# B&R Automation Studio project CombinedLinenSoiledA9KAN (part 4)

#### zzuld_3Cyclic.ab
```automation-basic
PROGRAM _CYCLIC
   	(* cyclic program *)

	;Unloading Programs 3 - Search and give Destination (Using Bag)

	;----------------------------------------
	;Version 1.00 03/12/2005 D.J. First Issue
	;----------------------------------------
	;Init Sequence
	;-------------

	;Spare Step
	IF (UldStep = 0) THEN
		UldStep = 1
	ENDIF

	;UldStep 1	- Check no bags in Storage are allocated with a destination
	IF (UldStep = 1) THEN

		;Allow next Discharger to search
		R_TRIG(NOT Std.BagsWithDestinations,PLS)
		IF PLS THEN
			Discharger 	= (LastDischarger + 1)
			ScanCount 	= 0
		ENDIF

		;Set ScanCount as alternating Value 25 is about 5 seconds
		IF Std.BagsWithDestinations  OR (ScanCount = 1) THEN
			Discharger 	= (Discharger + 1)
			ScanCount 	= 0
		ENDIF

		ScanCount = (ScanCount + 1)

		IF ((Discharger > EndDischarger) OR (Discharger < StartDischarger))  THEN
			Discharger 	= StartDischarger
		ENDIF

		;Set discharger number in TestDischarger if required
		IF (TestDischarger > 0) THEN
			Discharger = TestDischarger
		ENDIF

		;Read Program Variables
		n = RegOffset[Discharger]

		ProgramStep 			= D[1 + n]
		ProgQtyComplete			= D[2 + n]
		AutoRecirculation 		= (D[1003] = 1)		;Use if Re-cirulation or Offgoing Batching Loop
		RecirculationMaxDepth 	= D[1004]

		ManualLine       		= D[7 + n]
		ManualBags       		= D[8 + n]
		StepsSearched			= D[9 + n]
		SkipIncompleteStep 		= (D[10 + n] = 1)
		AutoRepeat				= (D[11 + n] = 1)
		MixCategories 			= (D[12 + n] = 1)	;Batch must be same category?
		MixCustomers 			= (D[13 + n] = 1) 	;Batch must be same customer?
		NoBagAvailable			= (D[14 + n] = 1)	;Alarm 'No Bag Available'
		ProgramFinished			= (D[15 + n] = 1)	;Alarm 'Finished Program'
		ManualLineRecirc 		= D[1016]
		ManualBagsRecirc 		= D[1017]
		ProgramRunning			= (D[19 + n] = 1)	;Run from TrackView
		ExpressLine 			= D[20 + n]
		CustomerMode			= D[21 + n]			;Customer Mode 0 = Normal Manual, 1 = Reset Pointer on every step, 2 = Check all steps before changing
		ProgramReset			= (D[22 + n] = 1)	;Customer FIFO Reset

		DischargerReady			= Uld[Discharger].SDCReady
		DischargerSpaces		= Line[BufferLineNum[Discharger]].SpaceBIT
		RecircSpaces			= Line[BufferLineNum[EndDischarger + 1]].SpaceBIT

		IF (NOT Std.BagsWithDestinations AND (Discharger > 0)) THEN
			UldStep = 2
		ELSE
			;Allow program to skip blank steps when Bags Have Destinations
			UnusedStep		= (D[40 + n + ProgramStep] = 0) ;Bags = 0
			IF UnusedStep THEN
				UldStep = 15
			ENDIF
		ENDIF

		;If program is new then Clear Search Values
		IF ProgramReset THEN
			Uld[Discharger].FIFOCustomer 		= 0	;Clear Current Customer - FIFO Will allocate next
			Uld[Discharger].LastCustQtyComplete = 0	;Clear Last Quantity
			StepsSearched 						= 0	;Clear Steps Searched / Failed
			D[22 + n]	 						= 0 ;Clear Program Reset
			UldStep 							= 0	;Keep Unloading Step at 0 to allow Customer FIFO to allocate next Customer
		ENDIF

	ENDIF

	;UldStep 2	- Check for a Manual Re-circulation regardless of Discharger
	;			- Note will stop all unloading progrms if not ready
	IF (UldStep = 2) THEN
		IF ((ManualLineRecirc >= StartLineSearch) AND (ManualLineRecirc <= EndLineSearch) AND (ManualBagsRecirc > 0)) THEN
			IF Uld[EndDischarger + 1].SDCReady THEN
				UldStep = 21
			ELSE
				UldStep = 0
			ENDIF
		ELSE
			UldStep = 3
		ENDIF
	ENDIF

	;UldStep 3	- Check Discharger is Ready
	IF (UldStep = 3) THEN
		IF (DischargerReady AND ProgramRunning AND (DischargerSpaces > 0)) THEN
			UldStep = 4
		ELSE
			;If not ready then clear steps searched
			UldStep = 0
		ENDIF
	ENDIF

	;UldStep 4	- Check for a Manual Bags
	IF (UldStep = 4) THEN
		IF ((ManualLine >= StartLineSearch) AND (ManualLine <= EndLineSearch) AND (ManualBags > 0)) THEN
			UldStep = 22
		ELSE
			UldStep = 5
		ENDIF
	ENDIF

	;STEP 5	- Check Express Line
	IF (UldStep = 5) THEN
		IF (ExpressLine > 0) THEN
			ExpressBag  = Line[ExpressLine].FirstBag
		ENDIF
		IF ((Bag[ExpressBag].Cat > 0) AND (ExpressLine > 0) AND (Line[BufferLineNum[Discharger]].SpaceBIT > 0)) THEN
			UldStep = 23
		ELSE
			UldStep = 6
		ENDIF
	ENDIF

	;UldStep 6	- Check Program step
	IF (UldStep = 6) THEN

		;Check if UldStep Valid
		IF (ProgramStep < 1) OR (ProgramStep > 20) THEN
			ProgramStep = 1 					;Set to UldStep 1
			ProgQtyComplete = 0 				;Clear Qty Completed
			IF (CustomerMode = 1) THEN
				Uld[Discharger].FIFOCustomer = 0
			ENDIF
		ENDIF

		UldStep = 7

	ENDIF

	;UldStep 7 - Check for remaining bags on the current Step
	IF (UldStep = 7) THEN

		BatchSize 		= D[80 + n + ProgramStep]
		Quantity 		= D[40 + n + ProgramStep] ;* BatchSize ;Take bags * BatchSize
		BagsRemaining 	= (Quantity - ProgQtyComplete)

		IF ((BagsRemaining > 0) AND (BagsRemaining >= BatchSize)) THEN
			UldStep = 8
		ELSE
			UldStep = 15 ;Step Not Complete Or No Qty
		ENDIF

	ENDIF

	;UldStep 8 - Check the 'Batch' Will fit onto the Buffer
	IF (UldStep = 8) THEN

		BatchSize 		= D[80 + n + ProgramStep]

		IF (DischargerSpaces >= BatchSize) THEN
			UldStep = 9
		ELSE
			UldStep = 0
		ENDIF

	ENDIF

	;UldStep 9 - Set Search Values
	IF (UldStep = 9) THEN

		IF (PriorityLine = 0) THEN
			StartLine = (Uld[Discharger].DischargerStartLine + 1)
			IF ((StartLine < StartLineSearch) OR (StartLine > EndLineSearch)) THEN
				StartLine = StartLineSearch
			ENDIF
		ELSE
			StartLine = PriorityLine
		ENDIF

		SearchLine   = D[60 + n + ProgramStep]
		BatchSize    = D[80 + n + ProgramStep]

		SearchCat[1] = D[100 + n + ProgramStep]
		SearchCat[2] = D[120 + n + ProgramStep]
		SearchCat[3] = D[140 + n + ProgramStep]

		IF (CustomerMode = 0) THEN
			SearchCus[1] = D[181 + n]					;Manually Selected Customer
		ELSE
			SearchCus[1] = Uld[Discharger].FIFOCustomer ;Automatic FIFO Customer Selection
		ENDIF

		SearchSpaces = 0 ;Search Always starts with no spaces on the recirc

		UldStep = 10

	ENDIF

	;UldStep 10 - Search for Bag(s) could be modified to run over several scans to reduce its load on the PLC
	;			  To find the best pos using set RecircSpaces low increasing to max.
	IF (UldStep = 10) THEN

		LOOP FindBest = 1 TO 3 DO

			;Clear the Search Array and Set Depth Allowed 1 for upto 49 storage lines
			FoundLine = 0
			memset(ADR(FoundBag[0]),0,10)
			memset(ADR(LineDepthAllowed[0]),1,50)

			RecircSpacesRemain = SearchSpaces

			IF (FindBest = 1) THEN
				MatchCat1Cus1 = TRUE
				MatchCat2Cus1 = FALSE
				MatchCat3Cus1 = FALSE
			ELSE IF (FindBest = 2) THEN
				MatchCat1Cus1 = MixCategories
				MatchCat2Cus1 = TRUE
				MatchCat3Cus1 = FALSE
			ELSE
				MatchCat1Cus1 = MixCategories
				MatchCat2Cus1 = MixCategories
				MatchCat3Cus1 = TRUE
			ENDIF

			;Loop around all the storage lins row by row.
			LOOP CurrentDepth = 1 TO UnloadingMaxDepth DO ;Always search to max depth to check scan time

				CurrentLine = StartLine

				LOOP LinesSearched = StartLineSearch TO EndLineSearch DO ;Loop around each line

					CurrentBag = (Line[CurrentLine].FirstBag + (CurrentDepth - 1))

					;Search / Add
					;------------
					;For Unloading by line - If there is a bag on the line and the 1st Category = 0 then check Customer valid
					;eg if the 1st Cat and 1st Cus are set to 0 then this would set "CatCusValid" to TRUE but the line must also match
					;Unloading by Customer only cannot be done.

					CusValid = FALSE
					CatValid = FALSE

					;Check the Customer is valid
					IF (Bag[CurrentBag].Cus = SearchCus[1]) THEN
						CusValid = TRUE
					ELSE IF ((SearchCus[1] = 0) AND (CustomerMode = 0)) THEN ;Only Valid If Manual Customer Selection
						CusValid = TRUE
					ENDIF

					;Check the Category is valid
					IF (MatchCat1Cus1 AND (Bag[CurrentBag].Cat = SearchCat[1]) AND (SearchCat[1] > 0)) THEN
						CatValid = TRUE
					ENDIF
					IF (MatchCat2Cus1 AND (Bag[CurrentBag].Cat = SearchCat[2]) AND (SearchCat[2] > 0)) THEN
						CatValid = TRUE
					ENDIF
					IF (MatchCat3Cus1 AND (Bag[CurrentBag].Cat = SearchCat[3]) AND (SearchCat[3] > 0)) THEN
						CatValid = TRUE
					ENDIF
					;If Unloading by line and no Category is set then Set Valid
					IF ((Bag[CurrentBag].Cat > 0) AND (SearchCat[1] = 0) AND (SearchLine > 0)) THEN
						CatValid = TRUE
					ENDIF

					LineValid = ((SearchLine = CurrentLine) OR (SearchLine = 0))

					DepthValid	= ((LineDepthAllowed[CurrentLine] + RecircSpacesRemain) >= CurrentDepth)
					DepthValid2	= ((CurrentDepth <= RecirculationMaxDepth) OR NOT AutoRecirculation)

					IF (CatValid AND CusValid AND LineValid AND DepthValid AND DepthValid2) THEN

						IF (FoundBag[0] < BatchSize)  THEN
							FoundBag[0] = FoundBag[0] + 1
							x 			= FoundBag[0]
							FoundBag[x] = CurrentBag
							FoundLine	= CurrentLine

							;If bags need to go to recirc then dec
							IF (LineDepthAllowed[CurrentLine] < USINT(CurrentDepth)) THEN
								SpacesUsed 			= USINT(CurrentDepth) - LineDepthAllowed[CurrentLine]
								RecircSpacesRemain 	= (RecircSpacesRemain - SpacesUsed)
							ENDIF

							LineDepthAllowed[CurrentLine] = USINT(CurrentDepth + 1)

						ENDIF

					ENDIF

					;-------------
					;End of Search
					;-------------

					;If searching using priority line then start from the Discharger Start Line
					IF CurrentLine = PriorityLine THEN
						CurrentLine = (Uld[Discharger].DischargerStartLine)
					ENDIF

					;Set Next Line
					CurrentLine = (CurrentLine + 1)
					IF CurrentLine > EndLineSearch THEN
						CurrentLine = StartLineSearch
					ENDIF

					;If the new line = priority line then skip as its already been searched
					IF CurrentLine = PriorityLine THEN
						CurrentLine = (CurrentLine + 1)
						IF CurrentLine > EndLineSearch THEN
							CurrentLine = StartLineSearch
						ENDIF
					ENDIF

				ENDLOOP

			ENDLOOP

			EXITIF FoundBag[0] = BatchSize

		ENDLOOP				;Find Best

		;Check if the bags were found
		IF FoundBag[0] = BatchSize THEN
			UldStep = 14 	;Action Results
		ELSE IF (AutoRecirculation AND (SearchSpaces < RecircSpaces)) THEN
			;If recirculation - to find the best possible result inc the search spaces each scan
			;until total spaces searched
			SearchSpaces = (SearchSpaces + 1)
			UldStep = 10	;Try with more recirculation space
		ELSE
			UldStep = 15	;Search Failed
		ENDIF

	ENDIF

	;UldStep 14 - Search Valid give bags destinations, inc qty taken by batchsize
	IF (UldStep = 14) THEN

		LOOP Dest = 1 TO BatchSize DO
			Bag[FoundBag[Dest]].Dst = USINT(BufferLineNum[Discharger])
		ENDLOOP
		ProgQtyComplete = ProgQtyComplete + BatchSize	;Inc Qty Completed
		StepsSearched = 0 								;Clear the search failed UldStep counter
		NoBagAvailable = FALSE 							;No Bags Alarm (OFF)
		LastDischarger = Discharger

		IF AutoRecirculation THEN
			UldStep = 24		;Set Any Bags for Auto-Reirculation
		ELSE
			UldStep = 0
		ENDIF

		;Mode 2 Needs to keep the Qty completed for the next customer
		Uld[Discharger].LastCustQtyComplete = ProgQtyComplete

	ENDIF

	;UldStep 15 - Search Failed
	IF (UldStep = 15) THEN

		BatchSize 		= D[80 + n + ProgramStep]
		;Quantity 		= D[40 + n + ProgramStep] * BatchSize ;Take bags * BatchSize
		Quantity		= (D[40 + n + ProgramStep])
		BagsRemaining 	= (Quantity - ProgQtyComplete)
		UnusedStep		= (D[40 + n + ProgramStep] = 0) ;Bags = 0

		;Inc Steps searched counter
		IF (StepsSearched < 21) THEN
			StepsSearched = (StepsSearched + 1)
		ENDIF

		IF (CustomerMode = 0) THEN
			IF (BagsRemaining = 0) THEN
				UldStep = 16			;Try Next Step
			ELSE IF (SkipIncompleteStep OR UnusedStep) THEN
				UldStep = 16			;Try Next Step
			ELSE
				NoBagAvailable = TRUE 	;Set Alarm and Wait for Operator to change Program or More Bags
				UldStep = 0
			ENDIF
		ENDIF

		IF (CustomerMode = 1) THEN
			IF (BagsRemaining = 0) THEN
				UldStep = 16			;Try Next Step
			ELSE IF (NOT UnusedStep) THEN
				IF (Uld[Discharger].FIFONextCustomer > 0) THEN
					;Mode 1 Search again with the Next Customer Without Changing Step
					Uld[Discharger].FIFOCustomer = Uld[Discharger].FIFONextCustomer
					UldStep = 0
				ELSE
					;Last customer was not found reset FIFO position to 1 and keep searching
					Uld[Discharger].FIFOCustomer = 0 ;Reset the First Customer
					NoBagAvailable = TRUE
					UldStep = 0
				ENDIF
			ELSE IF (SkipIncompleteStep OR UnusedStep) THEN
				UldStep = 16			;Try Next Step
			ELSE
				NoBagAvailable = TRUE	;Set Alarm and Wait for Operator to change Program or More Bags
				UldStep = 0
			ENDIf
		ENDIF

		IF (CustomerMode = 2) THEN
			IF (BagsRemaining = 0) THEN
				UldStep = 16			;Try Next Step
			ELSE IF (StepsSearched = 21) THEN
				IF (Uld[Discharger].FIFONextCustomer > 0) THEN
					;Mode 2 Customer Change Only After 21 Steps Searched
					Uld[Discharger].FIFOCustomer = Uld[Discharger].FIFONextCustomer
					ProgQtyComplete = Uld[Discharger].LastCustQtyComplete
					StepsSearched = 0 ;FREI Use -1 to go to next step
					UldStep = 0
				ELSE
					;Last customer was not found reset FIFO position to 1 and keep searching
					Uld[Discharger].FIFOCustomer = 0 ;Reset the First Customer
					NoBagAvailable = TRUE
					StepsSearched = 0
					UldStep = 0
				ENDIF
			ELSE IF (SkipIncompleteStep OR UnusedStep) THEN
				UldStep = 16			;Try Next Step
			ELSE
				NoBagAvailable = TRUE	;Set Alarm and Wait for Operator to change Program or More Bags
				UldStep = 0
			ENDIF
		ENDIF

	ENDIF

	;Skip Program Step or Set to 1
	IF (UldStep = 16) THEN
		IF (ProgramStep = 20) THEN
			IF AutoRepeat THEN
				ProgramStep = 1
				IF (CustomerMode = 1) THEN
					Uld[Discharger].FIFOCustomer = 0 ;Start Search With First Customer
				ENDIF
			ELSE
				ProgramFinished = TRUE
			ENDIF
		ELSE
			ProgramStep = ProgramStep + 1
			IF (CustomerMode = 1) THEN
				Uld[Discharger].FIFOCustomer = 0 ;Start Search With First Customer
			ENDIF
		ENDIF
		ProgQtyComplete = 0
		UldStep = 0
	ENDIF

	;UldStep 21 -	Manual Bags Recirc
	IF (UldStep = 21) THEN

		CurrentBag = Line[ManualLineRecirc].FirstBag

		IF Bag[CurrentBag].Cat > 0 THEN
			Bag[CurrentBag].Dst = USINT(BufferLineNum[EndDischarger + 1])	;Set Destination
			ManualBagsRecirc    = (ManualBagsRecirc - 1)					;Dec manual bags by 1
		ENDIF

		UldStep = 0

	ENDIF

	;UldStep 21 - Manual Bags to Discharger
	IF (UldStep = 22) THEN

		CurrentBag = Line[ManualLine].FirstBag

		IF Bag[CurrentBag].Cat > 0 THEN
			Bag[CurrentBag].Dst = USINT(BufferLineNum[Discharger])
			ManualBags 			= (ManualBags - 1)				;Dec manual bags by 1
		ENDIF

		UldStep = 0

	ENDIF

	;UldStep 23 - Express Line
	IF (UldStep = 23) THEN

		Bag[ExpressBag].Dst = USINT(BufferLineNum[Discharger])

		UldStep = 0

	ENDIF

	;UldStep 24 - Set Bags to re-circulation line if they need to move out of the way of bags with destinations
	IF (UldStep = 24) THEN

		LOOP CurrentLine = StartLineSearch to EndLineSearch DO
			LOOP CurrentBag = Line[CurrentLine].LastBag DOWNTO Line[CurrentLine].FirstBag DO

				IF (Bag[CurrentBag].Dst > 0) AND (Bag[CurrentBag - 1].Dst = 0) AND (CurrentBag > Line[CurrentLine].FirstBag) THEN
					Bag[CurrentBag - 1].Dst = USINT(BufferLineNum[EndDischarger + 1])
				ENDIF

			ENDLOOP
		ENDLOOP

		UldStep = 0

	ENDIF

	;Outputs
	;-------

	D[1 + n] 		= ProgramStep
	D[2 + n]		= ProgQtyComplete
	D[8 + n] 		= ManualBags
	D[9 + n]		= StepsSearched

	;No bag available is displayed if 20 steps have been searched and program is running
	IF (NoBagAvailable AND ProgramRunning) THEN
		D[14 + n] = 1
		Alarm[Discharger + 100].On		= TRUE
		Alarm[Discharger + 100].Bag 	= 0
		Alarm[Discharger + 100].Name 	= almUldNoBag
		Alarm[Discharger + 100].Beacon	= FALSE
	ELSE
		D[14 + n]	= 0
	ENDIF

	;Program is only finished if on step 20 and Program Running
	IF (ProgramFinished AND ProgramRunning AND (ProgramStep = 20)) THEN
		D[15 + n]	= 1
		Alarm[Discharger + 100].On		= TRUE
		Alarm[Discharger + 100].Bag 	= 0
		Alarm[Discharger + 100].Name 	= almUldProgFinished
		Alarm[Discharger + 100].Beacon	= FALSE
	ELSE
		D[15 + n]	= 0
	ENDIF

	;If no unloading alarms then clear unloading alarm
	IF (D[14 + n] = 0) AND (D[15 + n] = 0) THEN
		Alarm[Discharger + 100].On		= FALSE
		Alarm[Discharger + 100].Bag 	= 0
		Alarm[Discharger + 100].Name 	= almNoAlarm
		Alarm[Discharger + 100].Beacon	= FALSE
	ENDIF

	D[1017]		= ManualBagsRecirc

	IF ProgramRunning THEN
		D[18 + n]	= 1
	ELSE
		D[18 + n]	= 0
	ENDIF

	D[186 + n] 		= Uld[Discharger].FIFOCustomer
	D[187 + n] 		= Uld[Discharger].FIFONextCustomer

END_PROGRAM
```

### Program Logical/Sequences/can_drv2 (IEC, version 1.00.0) - * PowerTrans 1 & 2 NOT USED

#### can_drv2.var
```iecst
VAR RETAIN
	CAN_enable	:BOOL;
	ReadFrame1	:WET_CAN;
	EventRead1	:BOOL;
	EventWrite1	:BOOL;
	LastError	:UINT;
	n	:UINT;
	CANOK	:BOOL;
	WriteFrame1	:WET_CAN;
	EventRead2	:BOOL;
	EventWrite2	:BOOL;
	WriteFrame2	:WET_CAN;
END_VAR

VAR
	CANopen_01	:CANopen;
	DOInfo	:DatObjInfo;
	CANdftab_01	:CANdftab;
	error_var	:UDINT;
	data_adr	:UDINT;
	CANrwtab_01	:CANrwtab;
	EventWrite3	:BOOL;
	WriteFrame3	:WET_CAN;
	EventRead3	:BOOL;
END_VAR
```

#### can_drv2Init.ab
```automation-basic
PROGRAM _INIT
	(* init program *)

CAN_enable = 1
EventWrite1 = 0									;Reset CAN data table WRITE event
EventRead1 = 0  								;Reset CAN data table READ event
EventWrite2 = 0									;Reset CAN data table WRITE event
EventRead2 = 0  								;Reset CAN data table READ event
EventWrite3 = 0									;Reset CAN data table WRITE event
EventRead3 = 0  							    ;Reset CAN data table READ event

CANopen_01.enable		= CAN_enable
CANopen_01.baud_rate	= 25					;Define baud rate - 250 kbit/s
CANopen_01.cob_anz		= 100      				;Define number of link objects
CANopen_01.error_adr	= ADR(error_var)		;Define address for error output
CANopen_01.device		= ADR("SL3.SS1.IF3")	;Define number of device
CANopen_01.info			= 0

CANopen_01 FUB CANopen()						;Initiate CANopen

IF CANopen_01.status=0 THEN						;Check error level

	DOInfo.enable = 1
	DOInfo.pName  = "can_cmd"

	DOInfo FUB DatObjInfo()

	IF (DOInfo.status = 0) THEN

		data_adr					= DOInfo.pDatObjMem
		CANdftab_01.enable			= 1
		CANdftab_01.us_ident 		= CANopen_01.us_ident	;Set us_id
		CANdftab_01.table_adr		= data_adr				;Define address of data object
		CANdftab_01.tab_num			= UINT(DOInfo.len / 72)	;Define number of values

		CANdftab_01 FUB CANdftab()    						;Initiate CANdftab

		IF CANdftab_01.status = 0 THEN
			WriteFrame1.ControlSignals = BIT_SET(WriteFrame1.ControlSignals,0);Set Live Signal
			WriteFrame2.ControlSignals = BIT_SET(WriteFrame2.ControlSignals,0)
			WriteFrame3.ControlSignals = BIT_SET(WriteFrame3.ControlSignals,0)
			CANOK = TRUE
		ENDIF

	ENDIF

ENDIF
END_PROGRAM
```

#### can_drv2Cyclic.ab
```automation-basic
PROGRAM _CYCLIC
;----------------------------------------
;Version 1.00 08/02/2005 D.J. First Issue
;----------------------------------------

IF CANOK THEN

	;----------------
	;Set Write values
	;----------------

	;Powertrans 1
	IF CAN[1].BagReady THEN
		WriteFrame1.ControlSignals = BIT_SET(WriteFrame1.ControlSignals, 1)
	ELSE
		WriteFrame1.ControlSignals = BIT_CLR(WriteFrame1.ControlSignals, 1)
	ENDIF
	IF CAN[1].DoubleLoad THEN
		WriteFrame1.ControlSignals = BIT_SET(WriteFrame1.ControlSignals, 2)
	ELSE
		WriteFrame1.ControlSignals = BIT_CLR(WriteFrame1.ControlSignals, 2)
	ENDIF
	WriteFrame1.Destination = 0
	WriteFrame1.Category 	= CAN[1].Category
	WriteFrame1.Customer    = CAN[1].Customer
	WriteFrame1.Weight      = CAN[1].Weight

	;Write to Machine1
	EventWrite1 = TRUE

	;Powertrans 2
	;IF CAN[2].BagReady THEN
		;WriteFrame2.ControlSignals = BIT_SET(WriteFrame2.ControlSignals, 1)
	;ELSE
		;WriteFrame2.ControlSignals = BIT_CLR(WriteFrame2.ControlSignals, 1)
	;ENDIF
	;IF CAN[2].LoadFinished THEN
		;WriteFrame2.ControlSignals = BIT_SET(WriteFrame2.ControlSignals, 2)
	;ELSE
		;WriteFrame2.ControlSignals = BIT_CLR(WriteFrame2.ControlSignals, 2)
	;ENDIF
	;WriteFrame2.Destination = 0
	;WriteFrame2.Category 	= CAN[2].Category
	;WriteFrame2.Customer    = CAN[2].Customer
	;WriteFrame2.Weight      = CAN[2].Weight

	;Write to Machine2
	;EventWrite2 = TRUE

	;Powertrans 3
	;IF CAN[3].BagReady THEN
		;WriteFrame3.ControlSignals = BIT_SET(WriteFrame3.ControlSignals, 1)
	;ELSE
		;WriteFrame3.ControlSignals = BIT_CLR(WriteFrame3.ControlSignals, 1)
	;ENDIF
	;IF CAN[3].LoadFinished THEN
		;WriteFrame3.ControlSignals = BIT_SET(WriteFrame3.ControlSignals, 2)
	;ELSE
		;WriteFrame3.ControlSignals = BIT_CLR(WriteFrame3.ControlSignals, 2)
	;ENDIF
	;WriteFrame3.Destination = 0
	;WriteFrame3.Category 	= CAN[3].Category
	;WriteFrame3.Customer    = CAN[3].Customer
	;WriteFrame3.Weight      = CAN[3].Weight

	;Write to Machine3
	;EventWrite3 = TRUE

	;-----------------
	;Service CAN table
	;-----------------

	IF CANdftab_01.status=0 THEN						(*check error level*)
		CANrwtab_01.enable		= 1
		CANrwtab_01.tab_ident	= CANdftab_01.tab_ident (*define tab_id*)
		CANrwtab_01 FUB CANrwtab()						(*initiate CANrwtab*)
		LastError = CANrwtab_01.status
	ENDIF

	;----------------------------------
	;Check for incomming data from CBW1
	;----------------------------------

	;Powertrans 1
	IF EventRead1 THEN

		EventRead1 = FALSE

		CAN[1].Live 		  = BIT_TST(ReadFrame1.ControlSignals,0)
		CAN[1].DropLoad 	  = BIT_TST(ReadFrame1.ControlSignals,1)
		CAN[1].LoadDropped    = BIT_TST(ReadFrame1.ControlSignals,2)

		IF CAN[1].Live THEN
			CAN[1].LiveTime = 50	;5 seconds
		ENDIF

	ENDIF

	;----------------------------------
	;Check for incomming data from CBW1
	;----------------------------------

	;Powertrans 2
	;IF EventRead2 THEN

		;EventRead2 = FALSE

		;CAN[2].Live 		  = BIT_TST(ReadFrame2.ControlSignals,0)
		;CAN[2].DropLoad 	  = BIT_TST(ReadFrame2.ControlSignals,1)
		;CAN[2].LoadDropped    = BIT_TST(ReadFrame2.ControlSignals,2)
		;CAN[2].ReadyToLoad    = BIT_TST(ReadFrame2.ControlSignals,3)

		;IF CAN[2].Live THEN
			;CAN[2].LiveTime = 50	;5 seconds
		;ENDIF

	;ENDIF

	;----------------------------------
	;Check for incomming data from CBW1
	;----------------------------------

	;Powertrans 2
	;IF EventRead3 THEN

		;EventRead3 = FALSE

		;CAN[3].Live 		  = BIT_TST(ReadFrame3.ControlSignals,0)
		;CAN[3].DropLoad 	  = BIT_TST(ReadFrame3.ControlSignals,1)
		;CAN[3].LoadDropped    = BIT_TST(ReadFrame3.ControlSignals,2)
		;CAN[3].ReadyToLoad    = BIT_TST(ReadFrame3.ControlSignals,3)

		;IF CAN[3].Live THEN
			;CAN[3].LiveTime = 50	;5 seconds
		;ENDIF

	;ENDIF

	;-------------------
	;CAN Live / Presence
	;-------------------

	LOOP n = 1 TO 1 DO

		IF (CAN[n].LiveTime > 0) THEN
			CAN[n].LiveTime = (CAN[n].LiveTime - 1)
		ENDIF

		CAN[n].Live = (CAN[n].LiveTime <> 0)

	ENDLOOP

ENDIF
END_PROGRAM
```

### Program Logical/Sequences/zzclrmem (IEC) - * Clear Permanent Memory

#### zzclrmemCyclic.ab
```automation-basic
PROGRAM _CYCLIC
(* cyclic program *)

;Clear All Data Registers

IF ClearMem THEN

	memset(pC, 						0, SIZEOF(C))
	memset(pD, 						0, SIZEOF(D))
	memset(pBag, 					0, SIZEOF(Bag))
	memset(ADR(ReportBuffer), 		0, SIZEOF(ReportBuffer))
	memset(ADR(ReportLoading), 		0, SIZEOF(ReportLoading))
	memset(ADR(ReportUnloading), 	0, SIZEOF(ReportUnloading))

	Dave = SIZEOF(ReportBuffer)

	ClearMem = FALSE

ENDIF
END_PROGRAM
```

### Program Logical/Sequences/zzstn_q (IEC, version 1.00.0) - * Stations into Q

#### zzstn_qCyclic.ab
```automation-basic
PROGRAM _CYCLIC
 	(* cyclic program *)

;Sorting Stations Into Q with provision for Pushbutton into Q
;------------------------------------------------------------

;Set "AutoMaticRelease" in "zzconst"
;Nothing to change!

;-------------------------------------------
;Revision 1.00 - 19/12/2005 D.J. First Issue
;-------------------------------------------

StnsInQ 	= FALSE
StnsToPurge = FALSE

LOOP z = 1 TO Std.MaxWeighstations DO

	n = z

	;Force to Single station for testing / monitoring
	IF TestStation > 0 THEN
		n = TestStation
	ENDIF

	ManualRelease 	= (D[800 + n] = 1)
	PurgeStation	= (D[800 + n] = 2)

	;For testing force valid weight values
	IF TestWeight > 0 THEN
		Stn[n].Weight = TestWeight
	ENDIF

	;If Current weight is less than the Min Release Weight or SP2 is set below the Min Release Weight or SP3 is set below the Min Release Weight
	ValidWeight = ((Stn[n].Weight > Std.MinReleaseWeight) AND (D[3800 + n] > Std.MinReleaseWeight) AND  (D[3900 + n] > Std.MinReleaseWeight))

	;Testing
	;ValidWeight = TRUE

	;SP1 Reached - Approaching Weight
	SP1Reached = (Stn[n].Weight > D[3700 + n])

	;SP2 Reached - At Release Weight
	SP2Reached = (Stn[n].Weight > D[3800 + n])

	;SP3 Reached - Over Weight
	SP3Reached = (Stn[n].Weight > D[3900 + n])

	;Manual Release from TrackView
	IF ManualRelease THEN
		IF (ValidWeight AND (NOT SP3Reached)) THEN
			Stn[n].ManualRelease = TRUE
		ELSE IF (ValidWeight AND Std.EnableOverUnderRelease) THEN ;Enable Release KeySwitch
			Stn[n].ManualRelease = TRUE
		ENDIF
		D[800 + n] = 0 ;Cancel the Manual Release
	ENDIF

	IF PurgeStation THEN
		StnsToPurge = TRUE
	ENDIF

	;Enter Station into Q
	StnIntoQ = FALSE
	IF (Std.AutoMaticRelease AND SP2Reached AND ValidWeight AND (NOT SP3Reached)) THEN
		StnIntoQ = TRUE
	ELSE IF ((NOT Std.AutoMaticRelease) AND Stn[n].ReleaseButton AND SP2Reached AND ValidWeight AND (NOT SP3Reached)) THEN
		StnIntoQ = TRUE
	ELSE IF ((NOT Std.AutoMaticRelease) AND Stn[n].ReleaseButton AND Std.EnableOverUnderRelease AND ValidWeight) THEN ;AND (SP3Reached = FALSE) THEN
		StnIntoQ = TRUE
	ELSE IF (Stn[n].ManualRelease AND ValidWeight) THEN
		StnIntoQ = TRUE
	ENDIF

	IF StnIntoQ THEN
		StnsInQ = TRUE
		IF (Stn[n].QTime < $7FFF) THEN ;Keep within Integer range for PC
			Stn[n].QTime = (Stn[n].QTime + 1)
		ENDIF
	ELSE
		Stn[n].QTime = 0
	ENDIF

	D[100 + n] = Stn[n].QTime ;Set the time in the Q for Use by PC

	Stn[n].LampOn = FALSE
	Stn[n].SP1	= FALSE
	Stn[n].SP2	= FALSE
	Stn[n].SP3	= FALSE
	Stn[n].CloseFlap = FALSE
	Stn[n].LampFlashFast = FALSE
	IF (BIT_TST(D[998],0) = 1) THEN ;LampTest
		Stn[n].SP2 = TRUE
		Stn[n].CloseFlap = TRUE
	ELSE IF SP3Reached THEN
		Stn[n].SP3 = TRUE
		Stn[n].LampFlashFast = TRUE
		Stn[n].CloseFlap = TRUE
	ELSE IF SP2Reached AND NOT SP3Reached THEN
		Stn[n].SP2 = TRUE
		Stn[n].LampOn
		Stn[n].CloseFlap = TRUE
	ELSE IF SP1Reached AND NOT SP3Reached THEN
		Stn[n].SP1 = TRUE
	ENDIF

ENDLOOP

Std.StnsInQ 	= StnsInQ
Std.StnsToPurge = StnsToPurge
END_PROGRAM
```

### Program Logical/Sequences/zzreport (IEC) - * Reports to Master PC

#### zzreport.var
```iecst
VAR RETAIN
	ReportID	:UINT;
END_VAR

VAR
	n	:UINT;
	ReportPointer	:UINT;
	MaxReportBuffer	:UINT;
	MaxReportLoading	:UINT;
	MaxReportUnloading	:UINT;
	TestUnloadingCat	:UINT;
	AddUnloading	:BOOL;
END_VAR
```

#### zzreportCyclic.ab
```automation-basic
PROGRAM _CYCLIC
	;Reports To Graphics  - No changes required!

	;-----------------------------------------
	;Revision 1.00 19/01/2006 First Issue D.J.
	;-----------------------------------------

	;ReportBuffer 0 used to clear report all Zero
	ReportBuffer[0].Cat = 0
	ReportBuffer[0].Cus = 0
	ReportBuffer[0].Wgt = 0
	ReportBuffer[0].Cnt = 0
	ReportBuffer[0].Stn = 0
	ReportBuffer[0].Mcn = 0

	;Report array sizes - see declerations
	MaxReportBuffer		= 197	;1 less than array allocation as Array 0 is used as Zero values
	MaxReportLoading 	= 49	;Normally at least MaxStations
	MaxReportUnloading 	= 9		;Normally at least MaxDischargers

	;Shuffle reports buffer
	ReportPointer		= 0 	;Reports Pointer

	LOOP n = 1 TO MaxReportBuffer DO

		IF ((ReportBuffer[n].Cat = 0) AND (n < MaxReportBuffer)) THEN
			ReportBuffer[n] 		= ReportBuffer[n + 1]
			ReportBuffer[n + 1] 	= ReportBuffer[0]
		ENDIF

		;Inc Reports Pointer
		IF (ReportBuffer[n].Cat > 0) THEN
			ReportPointer = (ReportPointer + 1)
		ENDIF

	ENDLOOP

	;Put loaded reports into reports buffer
	LOOP n = 1 TO MaxReportLoading DO
		IF ((ReportBuffer[ReportPointer + 1].Cat = 0) AND (ReportPointer < MaxReportBuffer)) THEN
			IF (ReportLoading[n].Cat > 0) THEN
				ReportBuffer[ReportPointer + 1] = ReportLoading[n]
				ReportLoading[n] 				= ReportBuffer[0]
				ReportPointer 					= (ReportPointer + 1)
			ENDIF
		ENDIF
	ENDLOOP

	;Put unloaded reports into reports buffer
	LOOP n = 1 TO MaxReportUnloading DO
		IF ((ReportBuffer[ReportPointer + 1].Cat = 0) AND (ReportPointer < MaxReportBuffer)) THEN
			IF ReportUnloading[n].Cat > 0 THEN
				ReportBuffer[ReportPointer + 1] = ReportUnloading[n]
				ReportUnloading[n] 				= ReportBuffer[0]
				ReportPointer 					= (ReportPointer + 1)
			ENDIF
		ENDIF
	ENDLOOP

	;Reports Read from Graphics D[63]
	;Generate Unique Report ID
	IF (D[63] = ReportID) THEN
		;Clear first report
		ReportBuffer[1] = ReportBuffer[0]
		;Inc Report ID
		ReportID = ReportID + 1
	ENDIF

	;Set Report ID to Valid Range
	IF ((ReportID < 1) OR (ReportID > 9999)) THEN
		ReportID = 1
	ENDIF

	;Make Report at front of Q ready for Graphics
	IF (ReportBuffer[1].Cat > 0) THEN	;Reports Waiting
		D[1] = 1
	ELSE
		D[1] = 0
	ENDIF
	D[2] = ReportBuffer[1].Cus ;D2 = Reports Customer
	D[3] = ReportBuffer[1].Cat ;D3 = Reports Category
	D[4] = ReportBuffer[1].Wgt ;D4 = Reports Weight
	D[5] = ReportBuffer[1].Cnt ;D5 = Reports Count
	D[6] = ReportBuffer[1].Stn ;D6 = Reports Station
	D[7] = ReportBuffer[1].Mcn ;D7 = Reports Machine
	D[8] = 0 ;D8 = Reports Batch Code
	D[9] = 0 ;D9 = Reports Customer High?
	D[10] = ReportID

	;---------------
	;Reports testing
	;---------------

	;Add unloading report
	IF (AddUnloading AND (TestUnloadingCat > 0)) THEN
		IF (ReportUnloading[1].Cat = 0) THEN
			ReportUnloading[1].Cat = TestUnloadingCat	;Category
			ReportUnloading[1].Cus = 20					;Customer
			ReportUnloading[1].Wgt = 500				;Weight
			ReportUnloading[1].Cnt = 0					;Count
			ReportUnloading[1].Stn = 0					;Station
			ReportUnloading[1].Mcn = 1					;Machine
		ENDIF
		AddUnloading = FALSE
	ENDIF
END_PROGRAM
```

### Program Logical/Sequences/zzalarms (IEC) - * Alarms - Messages and History

#### zzalarmsCyclic.ab
```automation-basic
PROGRAM _CYCLIC
	(* cyclic program *)

;-----------------------------------------------
;Alarm Messages with Screen position and history
;-----------------------------------------------

;------------------------------------------------
;Version 1.00 - 08/12/2005 First Issue D.J.
;Vesrion 2.00 - 17/10/2006 Added Alarm.Extra D.J.
;------------------------------------------------

;Note - Sequence must set the following
;Alarm[x].on
;Alarm[x].Bag - for the bag position where the alarm will appear
;Alarm[x].Name - for the message that will be displayed use constants strating "alm"
;Alarn[x].Extra - Extra data for Graphics to use ie. Line number with fault on offgoing storage

I_CancelAlarm 	= FALSE ;X[4].X16
I_EStop 		= NOT X[8].X16
I_MotorOverload = Std.MotorOverload
I_InverterFault = FALSE ;(X[3].X03 OR X[3].X04 OR X[3].X05 OR X[3].X06)

;--------------
;Alarm Messages
;--------------

IF I_EStop THEN
	Alarm[100].On	= TRUE
	Alarm[100].Bag 	= 0
	Alarm[100].Name	= almEmergencyStop
ELSE IF I_MotorOverload THEN
	Alarm[100].On	= TRUE
	Alarm[100].Bag 	= 0
	Alarm[100].Name	= almMotorOverload
ELSE IF I_InverterFault THEN
	Alarm[100].On	= TRUE
	Alarm[100].Bag 	= 0
	Alarm[100].Name	= almInverterFault
ELSE
	Alarm[100].On	= FALSE
	Alarm[100].Bag 	= 0
	Alarm[100].Name	= almNoAlarm
ENDIF

;Shuffle the Alarms List

AlarmCount 		= 0
BeaconInList 	= FALSE

LOOP n = 1 TO 10 DO

	;If Alarm not on anymore the clear from the list
	AlmNumber = D[200 + n]
	IF NOT Alarm[AlmNumber].On THEN
		D[200 + n] = 0
		D[210 + n] = 0
	ENDIF

	;Shuffle the list down
	IF (D[200 + n] = 0) AND (D[201 + n] > 0) AND (n <> 10) THEN
		D[200 + n] = D[201 + n]
		D[210 + n] = D[211 + n]
		D[201 + n] = 0
		D[211 + n] = 0
	ENDIF

	;Set InList for any alarm in the list
	Alarm[D[200 + n]].InList = TRUE

	;Calculate total alarms in the list
	IF D[200 + n] > 0 THEN
		AlarmCount = AlarmCount + 1
	ENDIF

	;Is the alarm beacon required?
	IF Alarm[AlmNumber].On AND Alarm[AlmNumber].Beacon THEN
		BeaconInList = TRUE
	ENDIF

ENDLOOP

;Cancel the alarm beacon
IF I_CancelAlarm THEN
	CancelBeacon = TRUE
ENDIF

;Cancel the CancelAlarm beacon if no alarm in the list requires the beacon
IF NOT BeaconInList THEN
	CancelBeacon = FALSE
ENDIF

;Look at each sequence alarm and if not in list then add to list if space
LOOP n = 1 TO 109 DO

	;If alarm active and a code has been given and not in the list and history is clear then add
	IF ((AlarmCount < 10) AND Alarm[n].On AND NOT Alarm[n].InList AND ((D[221] = 0) OR (n > 100))) THEN

		;If name not set then set to general
		IF (Alarm[n].Name = 0) THEN
			Alarm[n].Name = almGeneralSequence
		ENDIF

		D[210] 			= n
		BuildD220		= LSL(Alarm[n].Extra,8)
		BuildD220 		= BuildD220 + Alarm[n].Name
		D[220] 			= BuildD220

		;New alarm found requiring the beacon
		IF Alarm[n].Beacon THEN
			CancelBeacon = FALSE
		ENDIF

		;Store to History - if not Unloading Alarm
		IF (n <= 100) THEN
			D[221] 			= n				;Alarm Number (Seq)
			D[222]			= Alarm[n].Name	;Alarm Name / Message
			D[223] 			= D[223] + 1	;Alarm ID
			D[224]			= Alarm[n].Extra;Alarm Extra Data
			IF D[223] > 32000 THEN
				D[223] = 1
			ENDIF
		ENDIF

		;Inc Total Alarms
		AlarmCount = AlarmCount + 1

	ENDIF

	;Cancel All InList's - will be checked on the next scan
	Alarm[n].InList = FALSE

ENDLOOP

;Show Alarm position on the screen
IF D[201] > 0 THEN
	D[0] = Alarm[D[201]].Bag
ELSE
	D[0] = 0
ENDIF

UnloadingAlarm = Alarm[101].On OR Alarm[102].On OR Alarm[103].On OR Alarm[104].On

;Alarm Output - Unloading Alarm cannot be cancelled
Y[5].Y16 = ((BeaconInList AND NOT CancelBeacon) OR UnloadingAlarm)
;Y[4].Y15 = CancelAlarm
END_PROGRAM
```

### Program Logical/Sequences/can_live (IEC, version 1.00.0) - * CAN Live status 1-32 to TrackView

#### can_live.var
```iecst
VAR
	CANLive_1 : BIT_ENCODE;
	CANLive_2 : BIT_ENCODE;
	TEST : BOOL;
END_VAR
```

#### can_liveCyclic.ab
```automation-basic
PROGRAM _CYCLIC
(* cyclic program *)

;------------------------------------------
;CAN Live / Status indication to TrackView
;------------------------------------------

;-----------------------------------------
;Revision 1.00 24/11/2005 D.J. First Issue
;-----------------------------------------

;Move CAN Status to Registers

;1-16
CANLive_1.Input[0] = CAN[1].Live OR TEST
CANLive_1.Input[1] = CAN[2].Live OR TEST
CANLive_1.Input[2] = CAN[3].Live
CANLive_1.Input[3] = CAN[4].Live
CANLive_1.Input[4] = CAN[5].Live
CANLive_1.Input[5] = CAN[6].Live
CANLive_1.Input[6] = CAN[7].Live
CANLive_1.Input[7] = CAN[8].Live
CANLive_1.Input[8] = CAN[9].Live
CANLive_1.Input[9] = CAN[10].Live
CANLive_1.Input[10] = FALSE ;Box[1].Live
CANLive_1.Input[11] = FALSE ;Box[2].Live
CANLive_1.Input[12] = FALSE ;Box[3].Live
CANLive_1.Input[13] = FALSE ;Box[4].Live
CANLive_1.Input[14] = FALSE ;Box[5].Live
CANLive_1.Input[15] = FALSE ;Box[6].Live

CANLive_1 FUB BIT_ENCODE()

D[76] = CANLive_1.Output

;17-32
CANLive_2.Input[0] = FALSE ;Box[7].Live
CANLive_2.Input[1] = FALSE ;Box[8].Live
CANLive_2.Input[2] = FALSE ;Box[9].Live
CANLive_2.Input[3] = CAN[20].Live
CANLive_2.Input[4] = CAN[21].Live
CANLive_2.Input[5] = CAN[22].Live
CANLive_2.Input[6] = CAN[23].Live
CANLive_2.Input[7] = CAN[24].Live
CANLive_2.Input[8] = CAN[25].Live
CANLive_2.Input[9] = CAN[26].Live
CANLive_2.Input[10] = CAN[27].Live
CANLive_2.Input[11] = CAN[28].Live
CANLive_2.Input[12] = CAN[29].Live
CANLive_2.Input[13] = CAN[30].Live
CANLive_2.Input[14] = CAN[31].Live
CANLive_2.Input[15] = CAN[32].Live

CANLive_2 FUB BIT_ENCODE()

D[77] = CANLive_2.Output
END_PROGRAM
```

### Package Logical/Sequences/TB - Transfer Belt

### Program Logical/Sequences/TB/12_belt2 (IEC) - * STB2 Transfer Belt 2

#### 12_belt2.var
```iecst
VAR RETAIN
	MinBeltRunCV : UINT;
END_VAR
VAR
	MinBeltRun : BOOL;
	BeltClearET : TIME;
	BeltClear : BOOL;
	LinenDetectedET : TIME;
	LinenDetected : BOOL;
	n : UINT;
END_VAR
VAR RETAIN
	STEP : UINT;
END_VAR
VAR
	Step6ET : TIME;
END_VAR
VAR RETAIN
	LASTSTEP : UINT;
END_VAR
VAR
	PLS : BOOL;
	O_RunBelt : BOOL;
	RunBelt : BOOL;
	TimerAlarm : TON_10ms;
	I_PhotoBottom : BOOL;
	I_PhotoTop : BOOL;
	Bank : UINT;
	WeightValid : BOOL;
	WeightValue : INT;
	BeltRunTime : UINT;
	BeltAddTime : UINT;
	CountValue : INT;
	CountValid : BOOL;
	StnBag : UINT;
	I_Started : BOOL;
END_VAR
```

#### 12_belt2.ab
```automation-basic
PROGRAM _CYCLIC
 	(* cyclic program *)

;Sequence 2 - Transfer Belt 1 from Stations 1-20

;-----------------------------------------
;Revision 1.00 18/01/2006 D.J. First Issue
;-----------------------------------------

;Inputs and Outputs
;------------------

Bank 						= 2

I_Started					= (D[2] > 0)
I_PhotoBottom 				= FALSE ;X[8].X15
I_PhotoTop   				= FALSE ;X[8].X15

Request.TransferBelt[Bank]	= FALSE

O_RunBelt 					= FALSE

Alarm[12].Name 				= 0
Alarm[12].Bag				= 242
Alarm[12].Beacon			= TRUE
Alarm[12].Extra				= 0
Alarm[12].Time				= 5000

n = D[911] ;Selected Station

STEP = D[912]
;Setup Pulse contact
PLS = (STEP <> LASTSTEP)
LASTSTEP = STEP

;Step 0 - Disabled
IF STEP = 0 THEN
	;Disabled
ENDIF

;Step 1 - Check no stations are releasing
IF STEP = 1 THEN
	;Don't allow stations to release
	Ldg[Bank].EnableStnRelease = FALSE
	;No Station Releaseng and switched on
	IF ((D[911] = 0) AND I_Started) THEN
		IF (Bag[242].Cat = 0) THEN
			D[912] = 2 ;No Bag on belt
		ELSE
			D[912] = 4 ;Bag on belt
		ENDIF
	ENDIF
	Alarm[12].Name = almNoAlarm
ENDIF

;Step 2 - Enable Station search
IF STEP = 2 THEN

	;Check each station to see if a manual destination has been set
	LOOP n = Ldg[Bank].StartStn TO Ldg[Bank].EndStn DO

		StnBag = n + (Std.StationBagsStart[Bank] - 1)

		IF ((Bag[StnBag].Dst > 0) AND (Bag[StnBag].Dst < 99) AND I_Started) THEN ;Dest 99 = Empty Bag in station
			Stn[n].DestManual = Bag[StnBag].Dst
		ELSE
			Stn[n].DestManual = 0
		ENDIF
		;For pairing set number of spaces to search for
		Stn[n].SpacesRequired = 0 ;D[2000 + Bag[StnBag].Prg]

	ENDLOOP

	;Station Search
	IF ((Ldg[Bank].Search = 0) AND I_Started AND NOT Std.EStop) THEN
		Ldg[Bank].Search = 1
	ELSE IF ((Ldg[Bank].Search = 2) AND (Ldg[Bank].Found > 0))  THEN

		D[911] 	= Ldg[Bank].Found
		n 		= D[911]

		StnBag 	= n + (Std.StationBagsStart[Bank] - 1)

		;Clear the release button count if used
		Stn[n].ManualRelease 	= FALSE
		Stn[n].PBCount 			= 0

		;------Write Report------
		IF Std.StationReports  THEN

			IF (ReportLoading[n].Cat = 0) THEN

				;Check if anything has been added and current weight is not less than the previous
				WeightValue = Stn[n].Weight - INT(StnPrev[n].Wgt)
				WeightValid = (WeightValue > 0)

				;Check if anything has been added and current weight is not less than the previous
				CountValue = Stn[n].Count - INT(StnPrev[n].Cnt)
				CountValid = (CountValue > 0)

				IF (WeightValid OR CountValid) THEN

					;Ensure valid values as we report on either a weight or count change
					IF (WeightValue < 0) THEN
						WeightValue = 0
					ENDIF

					IF (CountValue < 0) THEN
						CountValue = 0
					ENDIF

					ReportLoading[n].Prg = Bag[StnBag].Prg 			;Program
					ReportLoading[n].Cat = Bag[StnBag].Cat			;Category
					ReportLoading[n].Cus = Bag[StnBag].Cus			;Customer
					ReportLoading[n].Wgt = UINT(WeightValue)		;Weight
					ReportLoading[n].Cnt = UINT(CountValue)			;Count
					ReportLoading[n].Stn = n         				;Station
					ReportLoading[n].Mcn = 0						;Machine
					ReportLoading[n].Bid = Bag[StnBag].Bid			;Batch ID
				ENDIF

			ENDIF

		ENDIF

		;Set Previous Cat and Cus to Current and Clear Weight and Count
		StnPrev[n].Prg 	= Bag[StnBag].Prg
		StnPrev[n].Cat 	= Bag[StnBag].Cat
		StnPrev[n].Cus 	= Bag[StnBag].Cus
		StnPrev[n].Wgt 	= 0
		StnPrev[n].Cnt 	= 0
		StnPrev[n].Bid 	= Bag[StnBag].Bid

		;Copy Station Data to Belt Bag
		Bag[242] 		= Bag[StnBag]			;Copy complete bag data
		Bag[242].Dst 	= USINT(Ldg[Bank].Line)	;Destination
		Bag[StnBag].Dst = 0 					;Reset Destination (Manual)

		;Clear Manual Release and Count
		Stn[n].ManualRelease 	= FALSE
		Stn[n].Count			= 0

		;If Stations are too close to the loading unit then jump to wait for loading unit
		IF (n >= 1) AND (n <= 4) THEN
			D[912] = 6
		ELSE
			BeltAddTime = (D[911] / 2)
			Ldg[Bank].EnableStnRelease = TRUE
			D[912] = 3
		ENDIF

		Alarm[12].Name = almNoAlarm

	ENDIF
ELSE
	Ldg[Bank].Search  	= 0 ;Clear Search if not on step 2
ENDIF

;Step 3
;Open Bag and Release to Belt Conveyor
IF STEP = 3 THEN
	O_RunBelt  = TRUE
	IF (I_PhotoBottom OR I_PhotoTop	OR Test.TransferBelt) THEN
		D[912] = 4
	ENDIF
	Alarm[12].Name = almPhotocellNotMade
ENDIF

;Step 4 - Skipped
IF STEP = 4 THEN
	O_RunBelt = TRUE
	D[912] = 5
	Alarm[12].Name = almNoAlarm
ENDIF

;Step 5 - Run belt until top photocell is made.
IF STEP = 5 THEN
	O_RunBelt = TRUE
	IF I_PhotoTop OR Test.TransferBelt THEN
		D[912] = 6
	ENDIF
	Alarm[12].Name = almPhotocellNotMade
ENDIF

;Step 6 - Wait for loading unit ready
TON_10ms((STEP = 6),10,RunBelt,Step6ET)
IF STEP = 6 THEN
	O_RunBelt = (NOT RunBelt AND Ldg[Bank].EnableStnRelease)
	IF Enable.TransferBelt[Bank] THEN
		D[912] = 7
	ENDIF
ENDIF

;Step 7 - Run Belt until linen detected for 1 second and Station has emptied
TON_10ms(((STEP = 7) AND I_PhotoTop),100,LinenDetected,LinenDetectedET)
IF STEP = 7 THEN
	O_RunBelt = TRUE
	Ldg[Bank].EnableStnRelease = TRUE ;Enable Station to Open bags if they haven't been already
	IF (LinenDetected OR Test.TransferBelt) THEN
		D[912] = 8
	ENDIF
	Alarm[12].Name = almPhotocellNotMade
ENDIF

;Step 8 - Run Belt until photocells clear for 5 seconds
TON_10ms(((STEP = 8) AND NOT I_PhotoBottom AND NOT I_PhotoTop AND NOT Std.EStop),500,BeltClear,BeltClearET)
IF STEP = 8 THEN
	O_RunBelt = TRUE
	IF (BeltClear AND MinBeltRun AND (D[911] = 0)) THEN
		D[912] = 9
	ENDIF
	IF NOT Std.EStop THEN
		IF I_PhotoBottom OR I_PhotoTop THEN
			Alarm[12].Name = almPhotocellBlocked
		ELSE IF (D[911] <> 0) THEN
			Alarm[12].Name = almStationNotClosed
		ELSE IF NOT MinBeltRun THEN
			Alarm[12].Name = almClearingBeltPleaseWait
		ENDIF
	ENDIF
ENDIF

;Note - Unitl the Station has closed the min belt run time won't start
;Note - Speed for Horozintal belt = 45m/min and Inclined 55m/min
BeltRunTime = (10 + BeltAddTime)
CTU((O_RunBelt AND Std.Clock1s AND (D[911] = 0) AND NOT Std.EStop),(STEP = 1),BeltRunTime,MinBeltRun,MinBeltRunCV)

;Step 9 - Check Stations Are Closed
IF STEP = 9 THEN
	;Move Belt bag to loading unit
	IF PLS AND ((Bag[244].Cat = 0) AND (Bag[242].Cat > 0)) THEN
		Bag[244] = Bag[242]
		Bag[242] = Bag[0]
	ENDIF
	IF (D[911] = 0) THEN
		D[912] = 1
	ENDIF
	Alarm[12].Name = almStationNotClosed
ENDIF

;Alarms
TimerAlarm.IN = NOT PLS AND (Alarm[12].Name > 0)
TimerAlarm.PT = Alarm[12].Time
TimerAlarm FUB TON_10ms()
Alarm[12].On = TimerAlarm.Q
Alarm[12].ET = TimerAlarm.ET

;Outputs
;Inform Station Sequences that the belt has been
Ldg[Bank].BeltHasRun = ((D[912] > 3) AND Ldg[Bank].EnableStnRelease)

Y[85].Y07 = O_RunBelt
END_PROGRAM
```

### Library Logical/Libraries/IecCheck (IEC)
Depends on: Sys_Lib, AsString

#### IecCheck.st - Implementation file
```iecst
(********************************************************************
 * COPYRIGHT -- HP
 ********************************************************************
 * Library: IecCheck
 * Author: treamsbottom
 * Created: November 13, 2013
 ********************************************************************
 * Implementation of library IecCheck
 ********************************************************************)

(* Check divisor for DINT and UDINT division *)
FUNCTION CheckDivDWord
	IF divisor=0 THEN
		CheckDivDWord:=1;
		MakeEntry(55555,divisor,'CheckDivDWord');
	ELSE
		CheckDivDWord:=divisor;
	END_IF
END_FUNCTION

(* Check divisor for INT and UINT division *)
FUNCTION CheckDivWord
	IF divisor=0 THEN
		CheckDivWord:=1;
		MakeEntry(55555,divisor,'CheckDivWord');
	ELSE
		CheckDivWord:=divisor;
	END_IF
END_FUNCTION

(* Check divisor for SINT and USINT division *)
FUNCTION CheckDivByte
	IF divisor=0 THEN
		CheckDivByte:=1;
		MakeEntry(55555,divisor,'CheckDivByte');
	ELSE
		CheckDivByte:=divisor;
	END_IF
END_FUNCTION

(* Check divisor for REAL division *)
FUNCTION CheckDivReal
	IF divisor=0 THEN
		CheckDivReal:=1;
		MakeEntry(55555,0,'CheckDivReal');
	ELSE
		CheckDivReal:=divisor;
	END_IF
END_FUNCTION

(* Check divisor for LREAL division *)
FUNCTION CheckDivLReal
	IF divisor=0 THEN
		CheckDivLReal:=1;
		MakeEntry(55555,0,'CheckDivLReal');
	ELSE
		CheckDivLReal:=divisor;
	END_IF
END_FUNCTION

(* Check range for array access *)
FUNCTION CheckBounds
	IF index < lower THEN
		CheckBounds := lower;
		MakeEntry(55555,index,'RangeCheck');
	ELSIF index > upper THEN
		CheckBounds := upper;
		MakeEntry(55555,index,'RangeCheck');
	ELSE
		CheckBounds := index;
	END_IF
END_FUNCTION

(* Check range for enumeration *)
FUNCTION CheckRange
	IF value < lower THEN
		CheckRange := lower;
		MakeEntry(55555,value,'ENUM-Check');
	ELSIF value > upper THEN
		CheckRange := upper;
		MakeEntry(55555,value,'ENUM-Check');
	ELSE
		CheckRange := value;
	END_IF
END_FUNCTION

(* Check range for subrange of signed data types *)
FUNCTION CheckSignedSubrange
	IF value < lower THEN
		CheckSignedSubrange := lower;
		MakeEntry(55555,value,'CheckSignedSubrange');
	ELSIF value > upper THEN
		CheckSignedSubrange := upper;
		MakeEntry(55555,value,'CheckSignedSubrange');
	ELSE
		CheckSignedSubrange := value;
	END_IF
END_FUNCTION

(* Check range for subrange of unsigned data types *)
FUNCTION CheckUnsignedSubrange
	IF value < lower THEN
		CheckUnsignedSubrange := lower;
		MakeEntry(55555,value,'CheckUnsignedSubrange');
	ELSIF value > upper THEN
		CheckUnsignedSubrange := upper;
		MakeEntry(55555,value,'CheckUnsignedSubrange');
	ELSE
		CheckUnsignedSubrange := value;
	END_IF
END_FUNCTION

(* Check address when reading dynamic variables *)
FUNCTION CheckReadAccess
	IF address=0 THEN
		(* TODO: Insert an appropriate code, see AutomationStudio help for further information *)
		MakeEntry(55555,address,'Read from NULL');
	END_IF

	CheckReadAccess:=0;
END_FUNCTION

(* Check address when writing dynamic variables *)
FUNCTION CheckWriteAccess
	IF address=0 THEN
		(* TODO: Insert an appropriate code, see AutomationStudio help for further information *)
		MakeEntry(55555,address,'Write to NULL');
	END_IF

	CheckWriteAccess:=0;
END_FUNCTION

(* Makes an entry (log book entry) in the error log book *)
FUNCTION MakeEntry
		status_name := ST_name(0,ADR(taskname),ADR(group));

		strcpy(ADR(out_text),ADR(text));
		strcat(ADR(out_text),ADR(' > in task > '));
  		strcat(ADR(out_text),ADR(taskname));
		MakeEntry := ADR(out_text);
		ERRxfatal(number,index,ADR(out_text));
END_FUNCTION
```

### Library Logical/Libraries/WETCAN2

#### WETCAN2.typ
```iecst
TYPE
	COB_ID120 : 	STRUCT
		bBereit : BOOL;
		bContainerUeberBeladetrichter : BOOL;
		bProgrammOderKategorie : BOOL;
		uiProgrammKategorie : UINT;
		bPostennummer : BOOL;
		udPostennummer : UDINT;
		usFehlernummer : USINT;
		bAuftragskennzeichen : BOOL;
		szAuftragskennzeichen : STRING[12];
		udKundennummer : UDINT;
		uiGewicht : UINT;
		bNotAusHF : BOOL;
		bDatenuebernahmeLift : BOOL;
		bSchiebeVorposition : BOOL;
		usEinlaufInSpeibahnNr : USINT;
		usAuslaufAusSpeibahnNr : USINT;
		usReserve1 : USINT;
		usReserve2 : USINT;
		a_usCustomize : ARRAY[0..6] OF USINT;
	END_STRUCT;
	COB_ID121 : 	STRUCT
		bBereit : BOOL;
		bSackOeffnen : BOOL;
		bSackLeerWeiter : BOOL;
		bFreigLiftBeschickungSpeibahn : BOOL;
		bNotAusPT : BOOL;
		usReserve1 : USINT;
		usReserve2 : USINT;
		usReserve3 : USINT;
		usReserve4 : USINT;
		usReserve5 : USINT;
		usReserve6 : USINT;
		usReserve7 : USINT;
		bSchiebesignalPT : BOOL;
		a_usCustomize : ARRAY[0..6] OF USINT;
	END_STRUCT;
	COB_ID122 : 	STRUCT
		bBereit : BOOL;
		bProgKat : BOOL;
		uiProgKat : UINT;
		udKundennummer : UDINT;
		uiGewicht : UINT;
		bPostennummer : BOOL;
		udPostennummer : UDINT;
		bAuftrKennz : BOOL;
		szAuftragskennzeichen : STRING[12];
		bPostenAufBelband : BOOL;
		bPostendatenGueltig : BOOL;
		bNotAusSackbeladung : BOOL;
		usFehlerNr : USINT;
		usZaehler : USINT;
		usReserve1 : USINT;
		usReserve2 : USINT;
		a_usCustomize : ARRAY[0..6] OF USINT;
	END_STRUCT;
	COB_ID123 : 	STRUCT
		bBereit : BOOL;
		bDatenBereitstellen : BOOL;
		bBeladesignal : BOOL;
		bNotAusPT : BOOL;
		usReserve1 : USINT;
		usReserve2 : USINT;
		usReserve3 : USINT;
		usReserve4 : USINT;
		usReserve5 : USINT;
		usReserve6 : USINT;
		usReserve7 : USINT;
		a_usCustomize : ARRAY[0..6] OF USINT;
	END_STRUCT;
	COB_ID201 : 	STRUCT
		bBereit : BOOL;
		bVorsignal : BOOL;
		bEntladesignal : BOOL;
		bKeineRueckgewinnung : BOOL;
		bProgrammOderKategorie : BOOL;
		uiProgrammKategorie : UINT;
		udPostennummer : UDINT;
		udKundennummer : UDINT;
		uiGewicht : UINT;
		bNotAusWM : BOOL;
		bFreigabeDesinfektion : BOOL;
		bTankIstLeer : BOOL;
		bFreigabeSpuelen : BOOL;
		bEndeDesinfektion : BOOL;
		usReserve1 : USINT;
		a_usCustomize : ARRAY[0..6] OF USINT;
	END_STRUCT;
	COB_ID209 : 	STRUCT
		bBereit : BOOL;
		bVorsignal : BOOL;
		bEntladesignal : BOOL;
		bKeineRueckgewinnung : BOOL;
		bProgrammOderKategorie : BOOL;
		uiProgrammKategorie : UINT;
		udPostennummer : UDINT;
		udKundennummer : UDINT;
		uiGewicht : UINT;
		bNotAusWetShuttle : BOOL;
		usReserve1 : USINT;
		usReserve2 : USINT;
		a_usCustomize : ARRAY[0..6] OF USINT;
	END_STRUCT;
	COB_ID211 : 	STRUCT
		bBereit : BOOL;
		bBeladebereit : BOOL;
		bSchiebeimpSpbPreXOR_WETShuttle : BOOL;
		bSchiebeimpulsErsteEntwaess : BOOL;
		bSchiebeimpulsZweiteEntwaess : BOOL;
		bAblassvZwangsoeffnErsteEnt : BOOL;
		bAblassvZwangsoeffnZweiteEnt : BOOL;
		bFehlerBelgewErtsteEntwaess : BOOL;
		bFehlerBelgewZweiteEntwaess : BOOL;
		usFehlerErsteEntwaess : USINT;
		usFehlerZweiteEntwaess : USINT;
		usFehlerWetShuttle : USINT;
		bNotAusEntwaessWetShuttle : BOOL;
		bStartDesinfektion : BOOL;
		bStartSpuelen : BOOL;
		bEndeSpuelen : BOOL;
		bReserve1 : BOOL;
		bReserve2 : BOOL;
		bReserve3 : BOOL;
		bReserve4 : BOOL;
		bReserve5 : BOOL;
		bReserve6 : BOOL;
		bReserve7 : BOOL;
		bReserve8 : BOOL;
		bReserve9 : BOOL;
		bReserve10 : BOOL;
		a_usCustomize : ARRAY[0..6] OF USINT;
		bSicherheitstuerPTPP : BOOL;
		bStartbefehlAnPT : BOOL;
	END_STRUCT;
	COB_ID219 : 	STRUCT
		bBereitEntwWetShuttle : BOOL;
		bBereitEntw : BOOL;
		bBeladebereit : BOOL;
		bSchiebeimpuls : BOOL;
		bHANDWetShuttleEntladen : BOOL;
		bFehlerBeladegewicht : BOOL;
		usFehlerEntw : USINT;
		usFehlerWetShuttle : USINT;
		bNotAusEntw : BOOL;
		usReserve1 : USINT;
		usReserve2 : USINT;
		usReserve3 : USINT;
		usReserve4 : USINT;
		usReserve5 : USINT;
		usReserve6 : USINT;
		a_usCustomize : ARRAY[0..6] OF USINT;
	END_STRUCT;
	COB_ID221 : 	STRUCT
		bBereit : BOOL;
		bPostendatenGueltig : BOOL;
		bUnglPostenKeineDPBelAmTrockner : BOOL;
		bTrocknerprogOderKategorie : BOOL;
		uiTrocknerprogKategorie : UINT;
		udPostennummer : UDINT;
		udKundennummer : UDINT;
		uiGewicht : UINT;
		bNotAusWM : BOOL;
		usReserve1 : USINT;
		usReserve2 : USINT;
		a_usCustomize : ARRAY[0..6] OF USINT;
	END_STRUCT;
	COB_ID231 : 	STRUCT
		bBereit : BOOL;
		usBeladungTrockner : USINT;
		usEntladungTrockner : USINT;
		usTransferZBvorTrockner : USINT;
		usTransferZBvorHFB : USINT;
		usFehlernummer : USINT;
		bNotAusVerbundEinzeltr : BOOL;
		usReserve1 : USINT;
		usReserve2 : USINT;
		a_usCustomize : ARRAY[0..6] OF USINT;
	END_STRUCT;
	COB_ID251_253_255_257 : 	STRUCT
		bBereit : BOOL;
		bNotAusVerbund : BOOL;
		bProgKat : BOOL;
		uiProgKat : UINT;
		udPostennummer : UDINT;
		udKundennummer : UDINT;
		uiGewicht : UINT;
		usZiel : USINT;
		bBeladeende : BOOL;
		usReserve1 : USINT;
		bSperreBereich : BOOL;
		a_usCustomize : ARRAY[0..6] OF USINT;
		bBeladestart : BOOL;
	END_STRUCT;
	COB_ID252_254_256_258 : 	STRUCT
		bBereit : BOOL;
		bNotAusSackbeladung : BOOL;
		bSackBereit : BOOL;
		usReserve1 : USINT;
		usReserve2 : USINT;
		usReserve3 : USINT;
		usReserve4 : USINT;
		usReserve5 : USINT;
		usReserve6 : USINT;
		usReserve7 : USINT;
		a_usCustomize : ARRAY[0..6] OF USINT;
		bSperreBereich : BOOL;
	END_STRUCT;
	COB_ID261 : 	STRUCT
		bBereit : BOOL;
		bBeladungBeendet : BOOL;
		bBeladungAktiv : BOOL;
		bSaugboxBelegt : BOOL;
		bNotHaltSaugbox : BOOL;
		uiMeldung : UINT;
		uiGewicht : UINT;
	END_STRUCT;
	COB_ID262 : 	STRUCT
		bBereit : BOOL;
		bSackBereit : BOOL;
		bEntladefreigabe : BOOL;
		bNotHaltSackspeicher : BOOL;
	END_STRUCT;
	COB_ID301bis304 : 	STRUCT
		bBereit : BOOL;
		bEntwaesserungEntlaedt : BOOL;
		bPostenInEntwaesserung : BOOL;
		bEntladestoerungAnPresse : BOOL;
		bSperreFahrbandVonZentrifuge : BOOL;
		bProgrammOderKategorie : BOOL;
		uiProgrammKategorie : UINT;
		udPostennummer : UDINT;
		udKundennummer : UDINT;
		uiGewicht : UINT;
		bBandlaufEntladeband : BOOL;
		bVorsignalEntladung : BOOL;
		bNotAusEntwaesserung : BOOL;
		usReserve1 : USINT;
		a_usCustomize : ARRAY[0..6] OF USINT;
		bLichtschrankeBandende : BOOL;
		bEntladeueberwachung : BOOL;
	END_STRUCT;
	COB_ID306 : 	STRUCT
		bBereit : BOOL;
		bAeroEntlaedt : BOOL;
		bPostenInAero : BOOL;
		bSperreFahrbandVonAero : BOOL;
		bProgrammOderKategorie : BOOL;
		uiProgrammKategorie : UINT;
		udPostennummer : UDINT;
		udKundennummer : UDINT;
		uiGewicht : UINT;
		bNotAusAero : BOOL;
		usReserve1 : USINT;
		usReserve2 : USINT;
		a_usCustomize : ARRAY[0..6] OF USINT;
		bUebergabestoerung : BOOL;
	END_STRUCT;
	COB_ID110 : 	STRUCT
		udPostennummer : UDINT;
		udKundennummer : UDINT;
		uiProgrammKategorie : UINT;
		uiGewicht : UINT;
		bBereit : BOOL;
		bEntladesignal : BOOL;
		bEntladebereit : BOOL;
		bUebergabestoerung : BOOL;
		bNotAusEntsander : BOOL;
		bProgrammOderKategorie : BOOL;
		Alignm1 : USINT;
		Alignm2 : USINT;
		a_usCustomize : ARRAY[0..6] OF USINT;
	END_STRUCT;
	COB_ID111 : 	STRUCT
		bBereit : BOOL;
		bEntladefreigabe : BOOL;
		bUebernahmestoerung : BOOL;
		bNotAusBeladeband : BOOL;
		a_usCustomize : ARRAY[0..6] OF USINT;
	END_STRUCT;
	COB_ID307 : 	STRUCT
		bBereit : BOOL;
		bEntladesignal : BOOL;
		bPostenAufBand : BOOL;
		bEntladestoerungBand : BOOL;
		bKundenwechsel : BOOL;
		bBandlaufEntladeband : BOOL;
		bProgrammKategorie : BOOL;
		bNotAusVerbund : BOOL;
		udPostennummer : UDINT;
		uiGewicht : UINT;
		uiProgrammKategorie : UINT;
		udKundennummer : UDINT;
		a_usCustomize : ARRAY[0..6] OF USINT;
	END_STRUCT;
	COB_ID311bis314 : 	STRUCT
		bBereit : BOOL;
		bBeladebereit : BOOL;
		bUebernahmestoerungVerbETAero : BOOL;
		bEntladelichtschrZentrifuge : BOOL;
		bNotAusETVerbAero : BOOL;
		usReserve1 : USINT;
		usReserve2 : USINT;
		usReserve3 : USINT;
		usReserve4 : USINT;
		usReserve5 : USINT;
		usReserve6 : USINT;
		usReserve7 : USINT;
		a_usCustomize : ARRAY[0..6] OF USINT;
		bSchutzgitterOffen : BOOL;
		bStartPresse : BOOL;
	END_STRUCT;
	COB_ID316 : 	STRUCT
		bBereit : BOOL;
		bBeladebereit : BOOL;
		bUebernahmestoerungVerbET : BOOL;
		bNotAusVerbET : BOOL;
		usReserve1 : USINT;
		usReserve2 : USINT;
		usReserve3 : USINT;
		usReserve4 : USINT;
		usReserve5 : USINT;
		usReserve6 : USINT;
		usReserve7 : USINT;
		a_usCustomize : ARRAY[0..6] OF USINT;
	END_STRUCT;
	COB_ID317 : 	STRUCT
		bBereit : BOOL;
		bBeladebereit : BOOL;
		bBeladeunterbrechung : BOOL;
		bUebernahmestoerung : BOOL;
		bQuittierungKundenwechsel : BOOL;
		bNotAusAero : BOOL;
		a_usCustomize : ARRAY[0..6] OF USINT;
	END_STRUCT;
	COB_ID351bis354 : 	STRUCT
		bBereit : BOOL;
		bAktPosFehler : BOOL;
		bAktPosWarnung : BOOL;
		bAktPosGesperrt : BOOL;
		usAktPos : USINT;
		bProgrammOderKategorie : BOOL;
		uiProgrammKategorie : UINT;
		udPostennummer : UDINT;
		udKundennummer : UDINT;
		uiGewicht : UINT;
		usReserve1 : USINT;
		a_usCustomize : ARRAY[0..6] OF USINT;
		bIdxPostenspeicher_1 : BOOL;
		bIdxPostenspeicher_2 : BOOL;
		bIdxPostenspeicher_4 : BOOL;
		bNotAusAero : BOOL;
	END_STRUCT;
	COB_ID361bis369 : 	STRUCT
		usStation : USINT;
		bProgrammOderKategorie : BOOL;
		uiProgrammKategorie : UINT;
		udPostennummer : UDINT;
		udKundennummer : UDINT;
		uiGewicht : UINT;
		usReserve1 : USINT;
		a_usCustomize : ARRAY[0..6] OF USINT;
		bBereit : BOOL;
	END_STRUCT;
	COB_ID371bis379 : 	STRUCT
		bDruckstatus : BOOL;
		usDruckerfehler : USINT;
		usStation : USINT;
		usReserve1 : USINT;
		usReserve2 : USINT;
		usReserve3 : USINT;
		usReserve4 : USINT;
		usReserve5 : USINT;
		a_usCustomize : ARRAY[0..6] OF USINT;
		bBereit : BOOL;
	END_STRUCT;
	COB_ID401bis419 : 	STRUCT
		bBereit : BOOL;
		bBeladeanforderung : BOOL;
		bEntladefreigabe : BOOL;
		bAnsteuerungSpeicherband : BOOL;
		bProgrammOderKategorie : BOOL;
		uiProgrammKategorie : UINT;
		udPostennummer : UDINT;
		udKundennummer : UDINT;
		uiGewicht : UINT;
		bNotAusVerbST : BOOL;
		bVorsignal : BOOL;
		bKippsperre : BOOL;
		usReserve1 : USINT;
		usReserve2 : USINT;
		bFreigabeFlusen : BOOL;
		a_usCustomize : ARRAY[0..6] OF USINT;
	END_STRUCT;
	COB_ID421bis439 : 	STRUCT
		bBereit : BOOL;
		bBeladebereit : BOOL;
		bBelaedt : BOOL;
		bEntladebereit : BOOL;
		bEntlade : BOOL;
		bTrocknet : BOOL;
		bHauptgeblaese : BOOL;
		bFlusenabsaugung : BOOL;
		bAbkuehlung : BOOL;
		bLichtschrSpeicherbandHinten : BOOL;
		bLichtschrSpeicherbandVorne : BOOL;
		bTemperatureinheit : BOOL;
		uiAbluftTemp : UINT;
		bEIN : BOOL;
		bStoerung : BOOL;
		uiRestzeit : UINT;
		bProgrammOderKategorie : BOOL;
		uiProgrammKategorie : UINT;
		udPostennummer : UDINT;
		udKundennummer : UDINT;
		uiGewicht : UINT;
		bNotAusTrockner : BOOL;
		bHand : BOOL;
		uiIRTemp : UINT;
		usReserve1 : USINT;
		a_usCustomize : ARRAY[0..6] OF USINT;
	END_STRUCT;
	COB_ID441bis459 : 	STRUCT
		uiTrocknerrestzeit : UINT;
		usReserve1 : USINT;
		usReserve2 : USINT;
		usReserve3 : USINT;
		usReserve4 : USINT;
		usReserve5 : USINT;
		bVorsignalFlusen : BOOL;
		bSaugbeladungAktiv : BOOL;
		bAnforderungFlusen : BOOL;
		a_usCustomize : ARRAY[0..6] OF USINT;
	END_STRUCT;
	COB_ID480 : 	STRUCT
		bBereit : BOOL;
		bNotAusAero : BOOL;
		bBeladebereit : BOOL;
		bBeladungAktiv : BOOL;
		bStoerung : BOOL;
		bBeladeanfHalbauto : BOOL;
		bBeladepause : BOOL;
		bBeladeabbruch : BOOL;
		bFreigabeBeladung : BOOL;
		bDurchschleusenStart : BOOL;
		bProgKat : BOOL;
		uiProgKat : UINT;
		udPostennummer : UDINT;
		udKundennummer : UDINT;
		uiGewicht : UINT;
		usReserve1 : USINT;
		bReserve1 : BOOL;
		bReserve2 : BOOL;
		bReserve3 : BOOL;
		bReserve4 : BOOL;
		bReserve5 : BOOL;
		bReserve6 : BOOL;
		bReserve7 : BOOL;
		bReserve8 : BOOL;
		bReserve9 : BOOL;
		a_usCustomize : ARRAY[0..6] OF USINT;
	END_STRUCT;
	COB_ID481 : 	STRUCT
		bBereit : BOOL;
		bNotAusAnlagenStrg : BOOL;
		bBeladeanfAuto : BOOL;
		bStoerung : BOOL;
		bAnlagenstrgHalbauto : BOOL;
		bAnlagenstrgAuto : BOOL;
		bPauseAktiv : BOOL;
		bDurchschleusen : BOOL;
		bFreigabeDurchschl : BOOL;
		bProgKat : BOOL;
		uiProgKat : UINT;
		uiGewicht : UINT;
		udKundennummer : UDINT;
		udPostennummer : UDINT;
		usReserve1 : USINT;
		bReserve1 : BOOL;
		bReserve2 : BOOL;
		bReserve3 : BOOL;
		bReserve4 : BOOL;
		bReserve5 : BOOL;
		bReserve6 : BOOL;
		bReserve7 : BOOL;
		bReserve8 : BOOL;
		bReserve9 : BOOL;
		bReserve10 : BOOL;
		a_usCustomize : ARRAY[0..6] OF USINT;
	END_STRUCT;
	InitCAN2PV : 	STRUCT
		pPVData : UDINT;
		uiCANID : UINT;
		usCommDirection : USINT;
		pEvVar : UDINT;
		iMode : INT;
	END_STRUCT;
	_CAN1 : 	STRUCT
		T_By0 : USINT;
		T_By1 : USINT;
		T_By2_By3 : UINT;
		T_By4_By5 : UINT;
		T_By6_By7 : UINT;
	END_STRUCT;
	_CAN2 : 	STRUCT
		T1_By0 : USINT;
		T1_By1 : USINT;
		T1_By2_By3 : UINT;
		T1_By4_By5 : UINT;
		T1_By6_By7 : UINT;
		T2_By0 : USINT;
		T2_By1 : USINT;
		T2_By2_By3 : UINT;
		T2_By4_By5 : UINT;
		T2_By6_By7 : UINT;
		T3_By0 : USINT;
		T3_By1 : USINT;
		T3_By2_By3 : UINT;
		T3_By4_By5 : UINT;
		T3_By6_By7 : UINT;
		T4_By0 : USINT;
		T4_By1 : USINT;
		T4_By2_By3 : UINT;
		T4_By4_By5 : UINT;
		T4_By6_By7 : UINT;
		T5_By0 : USINT;
		T5_By1 : USINT;
		T5_By2_By3 : UINT;
		T5_By4_By5 : UINT;
		T5_By6_By7 : UINT;
	END_STRUCT;
	_CAN2Read : 	STRUCT
		uiObjNr : UINT;
		ab_ByteArray : ARRAY[0..49] OF USINT;
		iNumberReceivedTels : INT;
		iNumberOfTels : INT;
	END_STRUCT;
	_CAN2Write : 	STRUCT
		CAN2 : _CAN2;
		bBusy : BOOL;
		iNumberOfTels : INT;
		iTelsSent : INT;
		uiCOB_ident : UINT;
		tTimeLastTelSent : TIME;
	END_STRUCT;
	_CANAccess : 	STRUCT
		CANMulQueue_q_ident : UDINT;
		CANMulOpen_us_ident : UDINT;
		CANopen_us_ident : UDINT;
	END_STRUCT;
	_DOAccess : 	STRUCT
		DO_us_ident : UDINT;
	END_STRUCT;
	_InitCAN2PV : 	STRUCT
		pPVData : UDINT;
		uiObjNr : UINT;
		usCommDirection : USINT;
		udCAN_q_ident : UDINT;
		pEvVar : UDINT;
		uiCOB_ident : UINT;
		bRunning : BOOL;
		iMode : INT;
	END_STRUCT;
	_InitCAN2Protocol : 	STRUCT
		AccessInitDO : _DOAccess;
		CAN2DObCount : UINT;
		CANAccess : _CANAccess;
		DoAccessCAN2Write : _DOAccess;
		iMode : INT;
		DOAccessCAN2Read : _DOAccess;
	END_STRUCT;
END_TYPE
```

#### WETCAN2.fun
```iecst
FUNCTION_BLOCK _GetNumberOfCan1Tels
	VAR_INPUT
		pPV : UDINT;
		uiObjNr : UINT;
	END_VAR
	VAR_OUTPUT
		iNumberOfCan1Tels : INT;
		iStatus : INT;
	END_VAR
	VAR
		LocalPV : ARRAY[0..31] OF USINT;
		byteTemp : USINT;
		szOsVersion : STRING[80];
		TARGETInfo_1 : TARGETInfo;
	END_VAR
END_FUNCTION_BLOCK

FUNCTION_BLOCK _SetCAN2COBTypeToCAN2Type
	VAR_INPUT
		p_InitCAN2PV : UDINT;
	END_VAR
	VAR_OUTPUT
		pCAN2Data : UDINT;
		iStatus : INT;
	END_VAR
	VAR
		LocalCAN2Data : _CAN2;
		Local_InitCAN2PV : _InitCAN2PV;
		LocByte4Str : ARRAY[0..11] OF USINT;
		udShr16 : UDINT;
		uiShl8 : UINT;
		LocalCOB_Typ_421bis439 : COB_ID421bis439;
		LocalCOB_Typ_120 : COB_ID120;
		LocalCOB_Typ_121 : COB_ID121;
		LocalCOB_Typ_201 : COB_ID201;
		LocalCOB_Typ_301 : COB_ID301bis304;
		LocalCOB_Typ_231 : COB_ID231;
		LocalCOB_Typ_221 : COB_ID221;
		LocalCOB_Typ_401bis419 : COB_ID401bis419;
		LocalCOB_Typ_306 : COB_ID306;
		LocalCOB_Typ_351 : COB_ID351bis354;
		LocalCOB_Typ_361bis369 : COB_ID361bis369;
		LocalCOB_Typ_371bis379 : COB_ID371bis379;
		LocalCOB_Typ_316 : COB_ID316;
		LocalCOB_Typ_311 : COB_ID311bis314;
		LocalCOB_Typ_211 : COB_ID211;
		LocalCOB_Typ_122 : COB_ID122;
		LocalCOB_Typ_209 : COB_ID209;
		LocalCOB_Typ_219 : COB_ID219;
		TARGETInfo_0 : TARGETInfo;
		szOSVersion : STRING[80];
		LocalCOB_Typ_251 : COB_ID251_253_255_257;
		LocalCOB_Typ_252 : COB_ID252_254_256_258;
		LocalCOB_Typ_480 : COB_ID480;
		LocalCOB_Typ_481 : COB_ID481;
		usTemp : USINT;
		LocalCOB_Typ_123 : COB_ID123;
		usT1By5Temp : USINT;
		LocalCOB_Typ_441bis459 : COB_ID441bis459;
		usTempBy2 : USINT;
		usTempBy3 : USINT;
		LocalCOB_Typ_307 : COB_ID307;
		LocalCOB_Typ_317 : COB_ID317;
		LocalCOB_Typ_261 : COB_ID261;
		LocalCOB_Typ_262 : COB_ID262;
		LocalCOB_Typ_354 : COB_ID351bis354;
		LocalCOB_Typ_352 : COB_ID351bis354;
		LocalCOB_Typ_353 : COB_ID351bis354;
		pLocByte4Str : REFERENCE TO ARRAY[0..11] OF USINT;
		LocalCOB_Typ_110 : COB_ID110;
		LocalCOB_Typ_111 : COB_ID111;
	END_VAR
END_FUNCTION_BLOCK

FUNCTION_BLOCK _SetCAN2TypeToCAN1Type
	VAR_INPUT
		pCAN2Data : UDINT;
		iTelegramIndex : UINT;
	END_VAR
	VAR_OUTPUT
		pCAN1Data : UDINT;
		iStatus : INT;
	END_VAR
	VAR
		LocalCAN2UniData : _CAN2;
		LocalCAN1Data : _CAN1;
	END_VAR
END_FUNCTION_BLOCK

FUNCTION_BLOCK _GetCANIDFromObjNr
	VAR_INPUT
		udObjNr : UDINT;
	END_VAR
	VAR_OUTPUT
		udCANID : UDINT;
		iStatus : INT;
	END_VAR
END_FUNCTION_BLOCK

FUNCTION_BLOCK _GetPVSize
	VAR_INPUT
		uiObjNr : UINT;
	END_VAR
	VAR_OUTPUT
		iCobLength : SINT;
		iStatus : INT;
	END_VAR
	VAR
		COBTyp_120 : COB_ID120;
		COBTyp_121 : COB_ID121;
		COBTyp_122 : COB_ID122;
		COB_Typ_201 : COB_ID201;
		COB_Typ_211 : COB_ID211;
		COB_Typ_221 : COB_ID221;
		COB_Typ_231 : COB_ID231;
		COB_Typ_301 : COB_ID301bis304;
		COB_Typ_311 : COB_ID311bis314;
		COB_Typ_306 : COB_ID306;
		COB_Typ_316 : COB_ID316;
		COB_Typ_401bis419 : COB_ID401bis419;
		COB_Typ_421bis439 : COB_ID421bis439;
		COB_Typ_351 : COB_ID351bis354;
		COB_Typ_361bis369 : COB_ID361bis369;
		COB_Typ_371bis379 : COB_ID371bis379;
		COB_Typ_209 : COB_ID209;
		COB_Typ_219 : COB_ID219;
		COBTyp_251 : COB_ID251_253_255_257;
		COBTyp_252 : COB_ID252_254_256_258;
		COBTyp_480 : COB_ID480;
		COBTyp_481 : COB_ID481;
		COBTyp_123 : COB_ID123;
		COB_Typ_441bis459 : COB_ID441bis459;
		COB_Typ_307 : COB_ID307;
		COB_Typ_317 : COB_ID317;
		COB_Typ_261 : COB_ID261;
		COB_Typ_262 : COB_ID262;
		COB_Typ_110 : COB_ID110;
		COB_Typ_111 : COB_ID111;
	END_VAR
END_FUNCTION_BLOCK

FUNCTION_BLOCK _SetCAN1TypeToByteArray
	VAR_INPUT
		a_usInByteArray : ARRAY[0..49] OF USINT;
		udCanID : UDINT;
		CAN1Data : _CAN1;
	END_VAR
	VAR_OUTPUT
		bDataValid : BOOL;
		a_usOutByteArray : ARRAY[0..49] OF USINT;
		uiStatus : UINT;
	END_VAR
	VAR
		uiShr8 : UINT;
		TARGETInfo_0 : TARGETInfo;
		szOSVersion : STRING[80];
		usTemp : USINT;
		uiTemp : UINT;
		bAKZ : BOOL;
		usTemp2 : USINT;
		uiTemp211 : UINT;
		usTemp211 : USINT;
	END_VAR
END_FUNCTION_BLOCK

FUNCTION_BLOCK _Seti386CAN2TypeToCAN1Type
	VAR_INPUT
		pCAN2Data : UDINT;
		iTelegramIndex : INT;
	END_VAR
	VAR_OUTPUT
		pCAN1Data : UDINT;
	END_VAR
	VAR
		LocalCAN1Data : _CAN1;
		LocalCAN2UniData : _CAN2;
		uiShiftUPPERWord : UINT;
		uiShiftLOWERWord : UINT;
		pLocalCAN2UniData : REFERENCE TO _CAN2;
	END_VAR
END_FUNCTION_BLOCK

FUNCTION_BLOCK _ConvertDataToi386
	VAR_INPUT
		uiObjNr : UINT;
		ByteArrayMotorola : ARRAY[0..49] OF USINT;
	END_VAR
	VAR_OUTPUT
		ByteArrayi386 : ARRAY[0..49] OF USINT;
	END_VAR
	VAR
		usTempByte : USINT;
	END_VAR
END_FUNCTION_BLOCK

FUNCTION_BLOCK CAN2RW
	VAR_INPUT
		pCAN2Init_ident : UDINT;
		enable : BOOL;
	END_VAR
	VAR_OUTPUT
		uiStatus : UINT;
	END_VAR
	VAR
		p_InitCAN2Protocol : UDINT;
		Local_InitCAN2Protocol : _InitCAN2Protocol;
		iLoopIdx : INT;
		Local_InitCAN2PV : _InitCAN2PV;
		DatObjRead_fromDOWrite : DatObjRead;
		DatObjWrite_toDOWrite : DatObjWrite;
		DatObjRead_fromDORead : DatObjRead;
		DatObjWrite_toDORead : DatObjWrite;
		tActTime : TIME;
		tDiffTime : UDINT;
		DatObjRead_fromInitDO : DatObjRead;
		LocalCAN2Write : _CAN2Write;
		_SetCAN2TypeToCAN1Type_0 : _SetCAN2TypeToCAN1Type;
		CANquwr_1 : CANquwr;
		_GetCANIDFromObjNr_0 : _GetCANIDFromObjNr;
		uiStatusEvVar : UINT;
		_SetCAN2COBTypeToCAN2Type_0 : _SetCAN2COBTypeToCAN2Type;
		LocalCAN2Read : _CAN2Read;
		uiLocalEvVar : UINT;
		CANrd_0 : CANrd;
		LocalCAN1Data : _CAN1;
		_GetPVSize_0 : _GetPVSize;
		LocalCAN2Copy : _CAN2;
		_SetCAN1TypeToByteArray_0 : _SetCAN1TypeToByteArray;
		iIdx : INT;
		bOverwritePV : BOOL;
		LocalCAN2ReadBak : _CAN2Read;
		TARGETInfo_0 : TARGETInfo;
		bIntel : BOOL;
		bMotorola : BOOL;
		pOSVersion : STRING[80];
		_Seti386CAN2TypeToCAN1Type_0 : _Seti386CAN2TypeToCAN1Type;
		_ConvertDataToi386_1 : _ConvertDataToi386;
		ab_ByteArrayi386Temp : ARRAY[0..49] OF USINT;
		iResIdx : INT;
		iTelsSendIdx : INT;
		iTempNumberOfTels : INT;
	END_VAR
END_FUNCTION_BLOCK

FUNCTION_BLOCK CAN2Init
	VAR_INPUT
		enable : BOOL;
		usUniqueIDCAN2Init : USINT;
		szCANInterface : STRING[80];
		pInitCAN2PV : UDINT;
		uiNumberOfCAN2COBs : UINT;
		doMemType : USINT;
	END_VAR
	VAR_OUTPUT
		uiStatus : UINT;
		pCAN2Init_ident : UDINT;
		CANopen_0 : CANopen;
	END_VAR
	VAR
		DatObjCreate_InitDO : DatObjCreate;
		p_InitCAN2Protocol : UDINT;
		DO_StartAdr : UDINT;
		DO_StatInfo : UINT;
		DO_Len : UDINT;
		DO_Memtype : USINT;
		DO_Option : UDINT;
		DO_ID : UDINT;
		zzDatObjInfo00000 : DatObjInfo;
		DO_ChangeDat : DATE_AND_TIME;
		iLoopIdx : INT;
		Local_InitCAN2Protocol : _InitCAN2Protocol;
		DatObjWrite_InitDO : DatObjWrite;
		pStartAdrDO : UDINT;
		ErrAdrNotInUse : UDINT;
		CANqueue_0 : CANqueue;
		Local_InitCAN2PV : _InitCAN2PV;
		DatObjCreate_WriteDO : DatObjCreate;
		pStartAdrDOCAN2Write : UDINT;
		DO_IDCAN2Write : UDINT;
		DatObjWrite_WriteDO : DatObjWrite;
		_SetCAN2COBTypeToCAN2Type_0 : _SetCAN2COBTypeToCAN2Type;
		zzDatObjInfo00001 : DatObjInfo;
		CAN2Write : _CAN2Write;
		pStartAdrDOCAN2Read : UDINT;
		DatObjCreate_ReadDO : DatObjCreate;
		DatObjWrite_ReadDO : DatObjWrite;
		CAN2Read : _CAN2Read;
		DO_IDCAN2Read : UDINT;
		zzDatObjInfo00002 : DatObjInfo;
		LocalInitCAN2PV : InitCAN2PV;
		iLoopIdxTemp : INT;
		_GetNumberOfCan1Tels_0 : _GetNumberOfCan1Tels;
		szInitDO : STRING[80];
		szInitDOInstanceNumber : STRING[80];
		usInitDOInstanceNumber : USINT;
		szCAN2WriteDO : STRING[80];
		szCAN2ReadDO : STRING[80];
	END_VAR
END_FUNCTION_BLOCK

FUNCTION_BLOCK _version
	VAR
		szVersion : STRING[80];
		uiBuild : UINT;
	END_VAR
END_FUNCTION_BLOCK

FUNCTION _swapUINT : UINT (* Internal use only - V3.2.0 *)
	VAR
		usHIGHERBYTE : USINT;
		usLOWERBYTE : USINT;
	END_VAR
	VAR_INPUT
		uiIn : UINT;
	END_VAR
END_FUNCTION
```
